// TIA Portal V18 export
FUNCTION_BLOCK "enc_no_change_in_time"   // FB6, FBD
{ S7_Optimized_Access := 'TRUE' }
VERSION : 0.1
// stored: AutoNumber true, IsIECCheckEnabled false, IsRetainMemResEnabled false, MemoryReserve 100, SetENOAutomatically false, UDAEnableTagReadback false
   VAR_INPUT
      pt : Time := T#1s;
      FWD : Bool;
      REV : Bool;
      POS : Real;
   END_VAR
   VAR_OUTPUT
      ER_FWD : Bool;
      ER_REV : Bool;
   END_VAR
   VAR
      going_fwd { ExternalAccessible := 'False'; ExternalVisible := 'False'; ExternalWritable := 'False'} : Bool;
      going_rev { ExternalAccessible := 'False'; ExternalVisible := 'False'; ExternalWritable := 'False'} : Bool;
      going_not { ExternalAccessible := 'False'; ExternalVisible := 'False'; ExternalWritable := 'False'} : Bool;
      mem : Real;
      t_fwd { S7_SetPoint := 'True'} : TON_TIME;
      t_rev { S7_SetPoint := 'True'} : TON_TIME;
   END_VAR
BEGIN

REGION Network 1
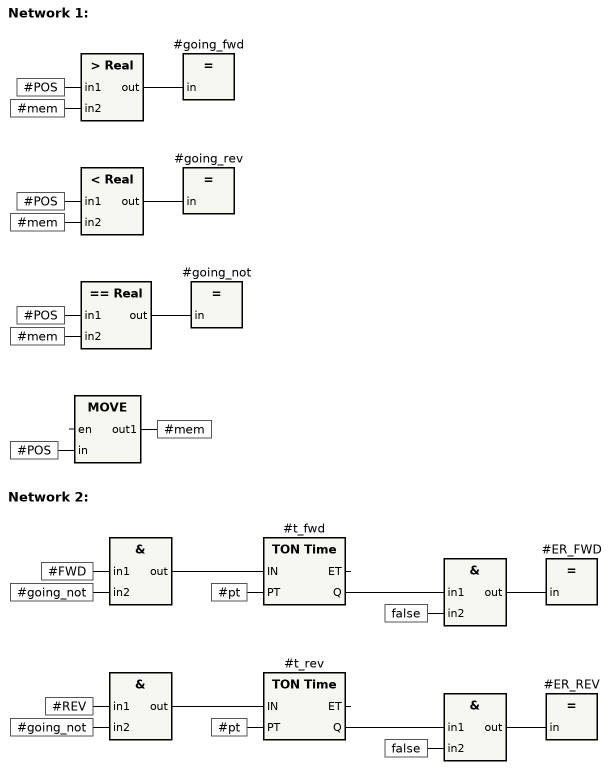
   #going_fwd := #POS > #mem;
   #going_rev := #POS < #mem;
   #going_not := #POS = #mem;
   #mem := #POS;
END_REGION

REGION Network 2
   #t_fwd(IN := #FWD AND #going_not, PT := #pt);   // TON
   #ER_FWD := #t_fwd.Q AND false;
   #t_rev(IN := #REV AND #going_not, PT := #pt);   // TON
   #ER_REV := #t_rev.Q AND false;
END_REGION
END_FUNCTION_BLOCK
